Staubli VAL3: OnEvent8.pgx

program OnEvent8()
  local bool l_bRes
begin
  //-----------------------------------------------------------------------
  //Header begin
  //LasMAN3.7
  //Description of program
  //
  //Input parameters
  //
  //Output paramaters
  //Example
  //  call OnEvent1()
  //History
  //  Creation : 2013-06-23  y.ye@staubli.com
  //Header end
  //-----------------------------------------------------------------------

  call UI:Control_YesNO("确定要退出吗?",l_bRes)
  if l_bRes
    bExit=true
  else
    DataBase:nInterfaceType=9
  endIf

end
